FUNCTION_BLOCK Z_TEMPERATURE2 (* Service Interface Function Block Type *)
  (* Standard: 61499-2; Function: Temperature sensor interface; Type: Service Interface Function Block; Description: Interface to a tsemperature sensor probe that samples a designated zone in the simulated environment. *)
  (* Version 1.0, 2020-01-04, badger, AUT, Original version *)
  (* Compiler header: #include Z_TEMPERATURE_Library.cpp. *)
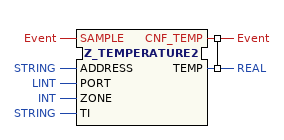
  EVENT_INPUT
    SAMPLE; (* Sample the environment to determine the latest zone temperature *)
  END_EVENT
  EVENT_OUTPUT
    CNF_TEMP WITH TEMP; (* Temperature is available *)
  END_EVENT
  VAR_INPUT
    ADDRESS : STRING := 127.0.0.1; (* URL of simulation server *)
    PORT : LINT := 62500; (* Listener port on the simulation server *)
    ZONE : INT := 1; (* Zone the temperature probe is sampling *)
    TI : STRING;
  END_VAR
  VAR_OUTPUT
    TEMP : REAL; (* The temperature measured by the probe *)
  END_VAR
  SERVICE APPLICATION/RESOURCE (* Service Interface Function Block Type *)
    SEQUENCE normal_establishment
      APPLICATION.INIT+(PARAMS) -> RESOURCE.initialize(PARAMS) -> APPLICATION.INITO+();
    END_SEQUENCE
    SEQUENCE unsuccessful_establishment
      APPLICATION.INIT+(PARAMS) -> RESOURCE.initialize(PARAMS) -> APPLICATION.INITO-(STATUS);
    END_SEQUENCE
    SEQUENCE request_confirm
      APPLICATION.REQ+(SD) -> RESOURCE.request(SD) -> APPLICATION.CNF+(RD);
    END_SEQUENCE
    SEQUENCE request_inhibited
      APPLICATION.REQ-(SD) -> APPLICATION.CNF-(STATUS);
    END_SEQUENCE
    SEQUENCE request_error
      APPLICATION.REQ+(SD) -> RESOURCE.request(SD) -> APPLICATION.CNF-(STATUS);
    END_SEQUENCE
    SEQUENCE indication_response
      RESOURCE.indicate(RD) -> APPLICATION.IND+(RD);
      APPLICATION.RSP(QI,SD) -> RESOURCE.response(QI,SD);
    END_SEQUENCE
    SEQUENCE indication_inhibited
      RESOURCE.indicate(RD,QI=FALSE) -> RESOURCE.inhibited();
    END_SEQUENCE
    SEQUENCE error_indication
      RESOURCE.error(STATUS) -> APPLICATION.IND-(STATUS);
    END_SEQUENCE
    SEQUENCE application_initiated_termination
      APPLICATION.INIT-() -> RESOURCE.terminate() -> APPLICATION.INITO-(STATUS);
    END_SEQUENCE
    SEQUENCE resource_initiated_termination
      -> APPLICATION.INITO-(STATUS);
    END_SEQUENCE
  END_SERVICE
END_FUNCTION_BLOCK
